TYPE Vec5d : ARRAY[1..5] OF LREAL; END_TYPE

(* stored: Version 1.1.0.1, ProductVersion 3.1.4024.12
   DUT Vec5d: Id {991e6e01-b87f-4cd9-af8d-0790583a537d} *)
